FUNCTION GetAnyType : __SYSTEM.AnyType
VAR_INPUT
	a		: ANY;
END_VAR
VAR
END_VAR

GetAnyType := a;

END_FUNCTION

(* stored: Version 1.1.0.1, ProductVersion 3.1.4024.11
   POU GetAnyType: Id {443949fb-0e92-45a1-919c-47897b524390}, SpecialFunc None *)
